(* CoDeSys 2.3.9.41 project: project_pump_station.pro *)
(* Libraries: STANDARD.LIB 4.10.05 11:14:46, IECSFC.LIB 13.4.06 15:51:28, SYSLIBTIME.LIB 26.10.21 13:46:42, SYSTASKINFO.LIB 26.10.21 13:46:42, ANALYZATION.LIB 5.10.99 09:05:06, Util.lib 18.5.10 15:14:28, SYSLIBCALLBACK.LIB 26.10.21 13:46:42 *)

(* PLC configuration (modules and I/O channels)
Fast discrete inputs [I_SIMPLE_INPUT] node 0, in %IB0 out %QB0 {ChannellName = Fast discrete inputs; Filtrationtime = 10000}
  AT %IX0.0 [BitInput] Discrete input 1 {ChannellName = Enter name}
  AT %IX0.1 [BitInput] Discrete input 2 {ChannellName = Enter name}
Discrete inputs [ID130] node 1, in %IB1 out %QB1 {ChannellName = Discrete inputs; Filtrationtime_GeneralINP = 16; PinCount = 16}
  discrete_input_first_byte AT %IB1.0 [ByteInput] discrete_input_first_byte {ChannellName = Enter name}
  discrete_input_second_byte AT %IB1.1 [ByteInput] discrete input_second_byte {ChannellName = Enter name}
Fast discrete outputs [OWEN_ID570] node 2, in %IB2 out %QB2 {ChannellName = Fast discrete outputs; SafeValueBool = FALSE; SafeValueBool = FALSE; SafeValueBool = FALSE; SafeValueBool = FALSE}
  hot_water_run_id1 AT %QX2.0 [BitOutput] Run hot water invertor drive1 {ChannellName = Enter name}
  hot_water_run_id2 AT %QX2.1 [BitOutput] Run hot water invertor drive2 {ChannellName = Enter name}
  water_supply_run_id1 AT %QX2.2 [BitOutput] Run water supply invertor drive1 {ChannellName = Enter name}
  water_supply_run_id2 AT %QX2.3 [BitOutput] Run water supply invertor drive2 {ChannellName = Enter name}
Discrete outputs [ID131] node 3, in %IB3 out %QB3 {ChannellName = Discrete outputs; SafeValueByte = 0; SafeValueByte = 0; SafeValueByteM = 0; PinCount = 24}
  AT %QB3.0 [ByteOutput] 8 discrete outputs {ChannellName = Enter name}
  AT %QB3.1 [ByteOutput] 8 discrete outputs {ChannellName = Enter name}
Special input [ID103] node 4, in %IB4 out %QB4 {ChannellName = Special input}
  AT %IX4.0 [BitInput] Special input {ChannellName = Enter name}
Special output [ID104] node 5, in %IB5 out %QB5 {ChannellName = Special output}
  AT %QX5.0 [BitOutput] Special output {ChannellName = Enter name}
ModBus (Master) [MODBUS_MASTER_ID450] node 6, in %IB6 out %QB6 {ChannellName = ModBus (Master); Visibility = No}
  AT %QD6.0 [DWordOutput] Last address {ChannellName = Enter name}
  AT %QW6.1 [WordOutput] Last error {ChannellName = Enter name}
  RS-485-1 [COM1_USART] node 0, in %IB6.0 out %QB6.0 {ChannellName = RS-485-1; CommunicationSpeed = 115200; Parity = NO PARITY CHECK; BitLength = 8 bits; StopLength = One stop bit; InterfaceType = RS485; FrameOriented = RTU; Timeout = 0; Visibility = No}
AT %QB6.1.0 [ComChannel] Command (0xff - Start) {ChannellName = Enter name}
Real input module [ID2007] node 0, in %IB6.1.0 out %QB6.1.0 {ChannellName = float input module; ModbusAddress = 4; Command_read_regs = Read holding Registers  (0x03); Visibility = No}
  input_pressure_hw AT %QD6.1.0.0 [FloatOutput] {ChannellName = Enter name}
Register input module [ID2003] node 1, in %IB6.1.1 out %QB6.1.1 {ChannellName = Register input module; ModbusAddress = 2; Command_read_regs = Read holding Registers  (0x03); Visibility = No}
  error_input_pressure_hw AT %QW6.1.1.0 [WordOutput] {ChannellName = Enter name}
Real input module [ID2007] node 2, in %IB6.1.2 out %QB6.1.2 {ChannellName = float input module; ModbusAddress = 10; Command_read_regs = Read holding Registers  (0x03); Visibility = No}
  output_pressure_hw AT %QD6.1.2.0 [FloatOutput] {ChannellName = Enter name}
Register input module [ID2003] node 3, in %IB6.1.3 out %QB6.1.3 {ChannellName = Register input module; ModbusAddress = 8; Command_read_regs = Read holding Registers  (0x03); Visibility = No}
  error_output_pressure_hw AT %QW6.1.3.0 [WordOutput] {ChannellName = Enter name}
Real input module [ID2007] node 4, in %IB6.1.4 out %QB6.1.4 {ChannellName = float input module; ModbusAddress = 16; Command_read_regs = Read holding Registers  (0x03); Visibility = No}
  input_pressure_ws AT %QD6.1.4.0 [FloatOutput] {ChannellName = Enter name}
Register input module [ID2003] node 5, in %IB6.1.5 out %QB6.1.5 {ChannellName = Register input module; ModbusAddress = 14; Command_read_regs = Read holding Registers  (0x03); Visibility = No}
  error_input_pressure_ws AT %QW6.1.5.0 [WordOutput] {ChannellName = Enter name}
Real input module [ID2007] node 6, in %IB6.1.6 out %QB6.1.6 {ChannellName = float input module; ModbusAddress = 22; Command_read_regs = Read holding Registers  (0x03); Visibility = No}
  output_pressure_ws AT %QD6.1.6.0 [FloatOutput] {ChannellName = Enter name}
Register input module [ID2003] node 7, in %IB6.1.7 out %QB6.1.7 {ChannellName = Register input module; ModbusAddress = 20; Command_read_regs = Read holding Registers  (0x03); Visibility = No}
  error_output_pressure_ws AT %QW6.1.7.0 [WordOutput] {ChannellName = Enter name}
AT %QD7.0 [DWordOutput] Last address {ChannellName = Enter name}
AT %QW7.1 [WordOutput] Last error {ChannellName = Enter name}
RS-485-1 [COM1_USART] node 0, in %IB7.0 out %QB7.0 {ChannellName = RS-485-1; CommunicationSpeed = 115200; Parity = NO PARITY CHECK; BitLength = 8 bits; StopLength = One stop bit; InterfaceType = RS485; FrameOriented = ASCII; Timeout = 0; Visibility = No}
Universal Modbus device [ID2000] node 1, in %IB7.1 out %QB7.1 {ChannellName = Universal Modbus device; ModuleIP = 10:0:0:223; ServiceTimeout = 150; TCPport = 502; NetMode = Serial; ModuleSlaveAddress = 1; RequestType = By poll time; PeriodOfService = 100; Visibility = No; RepeatCounter = 0; ByteSequence = Trace_mode}
  AT %QB7.1.0 [ComChannel] Command (0xff - Start) {ChannellName = Enter name}
output_value_hw_id1 AT %QW7.1.0.0 [WordOutput] {ChannellName = Enter name}
Register output module [ID2004] node 1, in %IB7.1.1 out %QB7.1.1 {ChannellName = Register; ModbusAddress = 0; Command_write_one_reg = Preset singl register (0x06); Visibility = No}
  output_value_hw_id2 AT %QW7.1.1.0 [WordOutput] {ChannellName = Enter name}
Register output module [ID2004] node 2, in %IB7.1.2 out %QB7.1.2 {ChannellName = Register; ModbusAddress = 0; Command_write_one_reg = Preset singl register (0x06); Visibility = No}
  output_value_ws_id1 AT %QW7.1.2.0 [WordOutput] {ChannellName = Enter name}
Register output module [ID2004] node 3, in %IB7.1.3 out %QB7.1.3 {ChannellName = Register; ModbusAddress = 0; Command_write_one_reg = Preset singl register (0x06); Visibility = No}
  output_value_ws_id2 AT %QW7.1.3.0 [WordOutput] {ChannellName = Enter name}
RS-232 [COM2_USART] node 0, in %IB8.0.0 out %QB8.0.0 {ChannellName = RS-232; CommunicationSpeed = 115200; Parity = NO PARITY CHECK; BitLength = 8 bits; StopLength = One stop bit; InterfaceType = RS232; FrameOriented = ASCII; Timeout = 0; Visibility = No}
8 bits [8Bit] node 1, in %IB8.1 out %QB8.1 {ChannellName = 8 bit}
  AT %QB8.1.0 [ByteOutput] {ChannellName = Enter name}
Float [Float] node 2, in %IB8.2 out %QB8.2 {ChannellName = float}
  hot_water_set_point_PID AT %QD8.2.0 [FloatOutput] {ChannellName = Enter name}
Float [Float] node 3, in %IB8.3 out %QB8.3 {ChannellName = float}
  water_supply_set_point_PID AT %QD8.3.0 [FloatOutput] {ChannellName = Enter name}
Float [Float] node 4, in %IB8.4 out %QB8.4 {ChannellName = float}
  P_hot_water AT %QD8.4.0 [FloatOutput] {ChannellName = Enter name}
Float [Float] node 5, in %IB8.5 out %QB8.5 {ChannellName = float}
  I_hot_water AT %QD8.5.0 [FloatOutput] {ChannellName = Enter name}
Float [Float] node 6, in %IB8.6 out %QB8.6 {ChannellName = float}
  D_hot_water AT %QD8.6.0 [FloatOutput] {ChannellName = Enter name}
Float [Float] node 7, in %IB8.7 out %QB8.7 {ChannellName = float}
  water_supply_P AT %QD8.7.0 [FloatOutput] {ChannellName = Enter name}
Float [Float] node 8, in %IB8.8 out %QB8.8 {ChannellName = float}
  water_supply_I AT %QD8.8.0 [FloatOutput] {ChannellName = Enter name}
Float [Float] node 9, in %IB8.9 out %QB8.9 {ChannellName = float}
  water_supply_D AT %QD8.9.0 [FloatOutput] {ChannellName = Enter name}
Float [Float] node 10, in %IB8.10 out %QB8.10 {ChannellName = float}
  hw_pressure_range_min AT %QD8.10.0 [FloatOutput] {ChannellName = Enter name}
Float [Float] node 11, in %IB8.11 out %QB8.11 {ChannellName = float}
  hw_pressure_range_max AT %QD8.11.0 [FloatOutput] {ChannellName = Enter name}
Float [Float] node 12, in %IB8.12 out %QB8.12 {ChannellName = float}
  water_supply_pressure_range_min AT %QD8.12.0 [FloatOutput] {ChannellName = Enter name}
Float [Float] node 13, in %IB8.13 out %QB8.13 {ChannellName = float}
  water_supply_pressure_range_max AT %QD8.13.0 [FloatOutput] {ChannellName = Enter name}
Float [Float] node 14, in %IB8.14 out %QB8.14 {ChannellName = float}
  hw_value_manual_frequency_id1 AT %QD8.14.0 [FloatOutput] {ChannellName = Enter name}
Float [Float] node 15, in %IB8.15 out %QB8.15 {ChannellName = float}
  hw_value_manual_frequency_id2 AT %QD8.15.0 [FloatOutput] {ChannellName = Enter name}
Float [Float] node 16, in %IB8.16 out %QB8.16 {ChannellName = float}
  water_supply_manual_frequency_id1 AT %QD8.16.0 [FloatOutput] {ChannellName = Enter name}
Float [Float] node 17, in %IB8.17 out %QB8.17 {ChannellName = float}
  water_supply_manual_frequency_id2 AT %QD8.17.0 [FloatOutput] {ChannellName = Enter name}
*)

(* Data type in Types data Analog_module/AnalogInputChannel *)
TYPE CAN_AnalogInputChannel :
STRUCT
	current_value: REAL;
	error_message: STRING(79);
END_STRUCT
END_TYPE

(* Data type in Types data SP310 *)
TYPE CAN_In_RS232_SP310 :
STRUCT
	pressure_input: REAL;
	pressure_output: REAL;
	status_run_invertor_drive1: BOOL;
	status_run_invertor_drive2: BOOL;
	status_alarm_invertor_drive1: BOOL;
	status_alarm_invertor_drive2: BOOL;
	PID_value: REAL;
END_STRUCT
END_TYPE

(* Data type in Types data Analog_module *)
TYPE CAN_in_RS485_Analog_module :
STRUCT

END_STRUCT
END_TYPE

(* Data type in Types data SP310 *)
TYPE CAN_Out_RS232_SP310 :
STRUCT
	auto_PID_enable: BOOL;
	cycle_enable: BOOL;
	cascade_enable: BOOL;
	set_point: REAL;
	P: REAL;
	I: REAL;
	D: REAL;
	value_manual_invertor_drive1: REAL;
	value_manual_invertor_drive2: REAL;
	pressure_range_min: REAL;
	pressure_range_max: REAL;

END_STRUCT
END_TYPE

(* Data type in ClassesProject/AnalogIModule/AnalogInputModule/AnalogInputChannel *)
TYPE classAnalogInputChannel :
STRUCT
	set_channel:classParamsValueScaling;
	value: REAL;
	error_code: WORD;
END_STRUCT
END_TYPE

(* Data type in ClassesProject/AnalogIModule/AnalogInputModule *)
TYPE classAnalogInputModule :
STRUCT
	channel1:classAnalogInputChannel;
	channel2:classAnalogInputChannel;
	channel3:classAnalogInputChannel;
	channel4:classAnalogInputChannel;
	channel5:classAnalogInputChannel;
	channel6:classAnalogInputChannel;
	channel7:classAnalogInputChannel;
	channel8:classAnalogInputChannel;
END_STRUCT
END_TYPE

(* Data type in ClassesProject/AnalogIModule/AnalogOutputModule/AnalogOutputChannel *)
TYPE classAnalogOutputChannel :
STRUCT
	register_value: WORD;
END_STRUCT
END_TYPE

(* Data type in ClassesProject/AnalogIModule/AnalogOutputModule *)
TYPE classAnalogOutputModule :
STRUCT
	channel1:classAnalogOutputChannel;
	channel2:classAnalogOutputChannel;
	channel3:classAnalogOutputChannel;
	channel4:classAnalogOutputChannel;
	channel5:classAnalogOutputChannel;
	channel6:classAnalogOutputChannel;
	channel7:classAnalogOutputChannel;
	channel8:classAnalogOutputChannel;
END_STRUCT
END_TYPE

(* Data type in ClassesProject/PLC_110_32_m2/DiscreteInputs/DiscreteInputByte *)
TYPE classDiscreteInputByte :
STRUCT
	Bit1:BOOL;
	Bit2:BOOL;
	Bit3:BOOL;
	Bit4:BOOL;
	Bit5:BOOL;
	Bit6:BOOL;
	Bit7:BOOL;
	Bit8:BOOL;
END_STRUCT
END_TYPE

(* Data type in ClassesProject/PLC_110_32_m2/DiscreteInputs *)
TYPE classDiscreteInputs :
STRUCT
	first_byte:classDiscreteInputByte;
	second_byte:classDiscreteInputByte;
END_STRUCT
END_TYPE

(* Data type in ClassesProject/PLC_110_32_m2/DiscreteOutputs/DiscreteOutputByte *)
TYPE classDiscreteOutputByte :
STRUCT
	Bit1:BOOL;
	Bit2:BOOL;
	Bit3:BOOL;
	Bit4:BOOL;
	Bit5:BOOL;
	Bit6:BOOL;
	Bit7:BOOL;
	Bit8:BOOL;
END_STRUCT
END_TYPE

(* Data type in ClassesProject/PLC_110_32_m2/DiscreteOutputs *)
TYPE classDiscreteOutputs :
STRUCT
	first_byte:classDiscreteOutputByte;
	second_byte:classDiscreteOutputByte;
END_STRUCT
END_TYPE

(* Data type in ClassesProject/PLC_110_32_m2/DiscreteInputs *)
TYPE classFastDiscreteInputs :
STRUCT
	Bit1:BOOL;
	Bit2:BOOL;
END_STRUCT
END_TYPE

(* Data type in ClassesProject/PLC_110_32_m2/DiscreteOutputs *)
TYPE classFastDiscreteOutputs :
STRUCT
	Bit1:BOOL;
	Bit2:BOOL;
	Bit3:BOOL;
	Bit4:BOOL;
END_STRUCT
END_TYPE

(* Data type in ClassesProject/InfoMessages/InfoAnalogInputModule/InfoAnalogInputChannel *)
TYPE classInfoAnalogInputChannel :
STRUCT
	current_value:REAL;
	measure:REAL;
	error_message:STRING(79);
END_STRUCT
END_TYPE

(* Data type in ClassesProject/InfoMessages/InfoAnalogInputModule *)
TYPE classInfoAnalogInputModule :
STRUCT
	channel1:classInfoAnalogInputChannel;
	channel2:classInfoAnalogInputChannel;
	channel3:classInfoAnalogInputChannel;
	channel4:classInfoAnalogInputChannel;
	channel5:classInfoAnalogInputChannel;
	channel6:classInfoAnalogInputChannel;
	channel7:classInfoAnalogInputChannel;
	channel8:classInfoAnalogInputChannel;
END_STRUCT
END_TYPE

(* Data type in ClassesProject/InfoMessages *)
TYPE classInfoCycle :
STRUCT
	run_timer: BOOL; (* статус работы таймера *)
	working_time: TIME; (*  время работы таймера *)
END_STRUCT
END_TYPE

(* Data type in ClassesProject/InfoMessages/InfoInvertorDrive *)
TYPE classInfoInvertorDrive :
STRUCT
	status_run:STRING(79);
	status_alarm:STRING(79);
	frequency:REAL;
END_STRUCT
END_TYPE

(* Data type in ClassesProject/InfoMessages *)
TYPE classInfoMessage :
STRUCT
	working_time: TIME;
	time_left: TIME;
END_STRUCT
END_TYPE

(* Data type in ClassesProject/InfoMessages/InfoPID *)
TYPE classInfoPid :
STRUCT
	out_value:REAL:=0;
	limits_active:BOOL:=FALSE;
	overflow:BOOL:=FALSE;
END_STRUCT
END_TYPE

(* Data type in ClassesProject/InvertorDrive *)
TYPE classInvertorDrive :
STRUCT
	discrete_inputs:classInvertorDriveDiscreteInputs;
	discrete_outputs:classInvertorDriveDiscreteOutputs;
	analog_input:classInvertorDriveAnalogInputs;
	analog_output:classInvertorDriveAnalogOutputs;
	set:classSetInvertorDrive;
	min_frequency:INT;
	max_frequency:INT;
	set_frequency:REAL;
	real_frequency:REAL;(* значение с аналогового выхода частотника *)
END_STRUCT
END_TYPE

(* Data type in ClassesProject/InvertorDrive *)
TYPE classInvertorDriveAnalogInputs :
STRUCT
	set_frequency:REAL;
END_STRUCT
END_TYPE

(* Data type in ClassesProject/InvertorDrive *)
TYPE classInvertorDriveAnalogOutputs :
STRUCT
	out_frequency:REAL;
END_STRUCT
END_TYPE

(* Data type in ClassesProject/InvertorDrive *)
TYPE classInvertorDriveDiscreteInputs :
STRUCT
	start:BOOL;
	reset_fault:BOOL;
END_STRUCT
END_TYPE

(* Data type in ClassesProject/InvertorDrive *)
TYPE classInvertorDriveDiscreteOutputs :
STRUCT
	status_run:BOOL;
	status_alarm:BOOL;
END_STRUCT
END_TYPE

(* Data type in ClassesProject/classesFunction *)
TYPE classParamsValueScaling :
STRUCT
	in_min: REAL:=0;
	in_max: REAL:=100;
	out_min: REAL:=0;
	out_max: REAL:=100;
END_STRUCT
END_TYPE

(* Data type in ClassesProject/PLC_110_32_m2 *)
TYPE classPLC110_32 :
STRUCT
	fast_discrete_inputs:classFastDiscreteInputs;
	discrete_inputs:classDiscreteInputs;
	special_input:classSpecialInput;
	fast_discrete_outputs:classFastDiscreteOutputs;
	discrete_output:classDiscreteOutputs;
	special_output:classSpecialOutput;
END_STRUCT
END_TYPE

(* Data type in ClassesProject/InfoMessages/PLC/110_32_m2 *)
TYPE classPLC32m2StatusInputs :
STRUCT
	fast_inputs:classFastDiscreteInputs;
	discrete_inputs:classDiscreteInputs;
	special_input:classSpecialInput;
END_STRUCT
END_TYPE

(* Data type in ClassesProject/InfoMessages/PLC/110_32_m2 *)
TYPE classPLC32m2StatusOutputs :
STRUCT
	fast_outputs:classFastDiscreteOutputs;
	discrete_outputs:classDiscreteOutputs;
	special_output:classSpecialOutput;
END_STRUCT
END_TYPE

(* Data type in ClassesProject/SP310/PumpStationSettings *)
TYPE classPumpStation :
STRUCT
	source:STRING(2);
	pump1:BOOL;
	pump2:BOOL;
	P:REAL;
	I:REAL;
	D:REAL;
	set_point:REAL;
	cycle_enable:BOOL;
	cascade_enable:BOOL;
	seconds_cycle: TIME;
	minutes_cycle: TIME;
	hours_cycle: TIME;
END_STRUCT
END_TYPE

(* Data type in ClassesProject/AnalogIModule/AnalogInputModule/SetAnalogInputsModule/SetAnalogInputChannel *)
TYPE classSetAnalogInputChannel :
STRUCT
	(* Конфигурационные параметры канала модуля. см. инструкцию прибора: приложение. таблица В.2 *)
	(* Границы АЦП и значения по умолчанию: для датчика 4-20mA  *)
	ain_l: REAL := 0;  (* Параметр Ain.L *)
	ain_h: REAL := 1000;  (* Параметр Ain.H *)
	analog_min_value: REAL := 4;  (* Диапазон нижней границы датчика давления *)
	analog_max_value: REAL := 20;  (* Диапазон верхней границы датчика давления *)
END_STRUCT
END_TYPE

(* Data type in ClassesProject/AnalogIModule/AnalogInputModule/SetAnalogInputsModule *)
TYPE classSetAnalogInputsModule :
STRUCT
	ch1_set:classSetAnalogInputChannel;
	ch2_set:classSetAnalogInputChannel;
	ch3_set:classSetAnalogInputChannel;
	ch4_set:classSetAnalogInputChannel;
	ch5_set:classSetAnalogInputChannel;
	ch6_set:classSetAnalogInputChannel;
	ch7_set:classSetAnalogInputChannel;
	ch8_set:classSetAnalogInputChannel;
END_STRUCT
END_TYPE

(* Data type in ClassesProject/InvertorDrive/SetInvertorDrive/SetAutoInvertorDrive *)
TYPE classSetAutoInvertorDrive :
STRUCT
	auto:BOOL:=FALSE;
	direct_logic:BOOL:=TRUE;  (* флаг прямого/обратного управления; при обратном управлении если значение контролируемой величины ниже уставки, выходная частота уменьшается, и наоборот*)
	set_point:REAL:=0;  (* уставка, задается в единицах измерения контролируемой величины *)
	value:REAL:=0;  (* текущее значение контролируемой величины, получаемое с датчика *)
	P:REAL:=2;  (* Пропорциональный коэффициент регулятора, при увеличении выход регулятора изменяется быстрее*)
	I:INT:=10;  (* Интегральный коэффичиент регулятора, время в секундах *)
	D:INT:=0;  (* Дифференциальный коэффичиент регулятора, время в секундах *)
END_STRUCT
END_TYPE

(* Data type in ClassesProject/InvertorDrive/SetInvertorDrive *)
TYPE classSetInvertorDrive :
STRUCT
	set_auto:classSetAutoInvertorDrive;
	set_frequency:classSetLimitFrequency;
END_STRUCT
END_TYPE

(* Data type in ClassesProject/Sensors/Kpi *)
TYPE classSetKpi :
STRUCT
	range:REAL;
	diff:REAL:=0.2;
END_STRUCT
END_TYPE

(* Data type in ClassesProject/InvertorDrive/SetInvertorDrive/SetLimitFrequency *)
TYPE classSetLimitFrequency :
STRUCT
	manual:REAL;  (* Hz *)
	min_range:REAL;  (* Hz *)
	max_range:REAL;  (* Hz *)
END_STRUCT
END_TYPE

(* Data type in ClassesProject/PID *)
TYPE classSetPid :
STRUCT
	actual:REAL;
	set_point:REAL;
	P:REAL;  (* Пропорциональный коэффициент регулятора, при увеличении выход регулятора изменяется быстрее*)
	I:INT;  (* Интегральный коэффичиент регулятора, время в секундах *)
	D:INT;  (* Дифференциальный коэффичиент регулятора, время в секундах *)
	Y_manual:REAL:=0;
	Y_offset:REAL;
	Y_min:REAL;
	Y_max:REAL;
	manual:BOOL;
	reset:BOOL;
END_STRUCT
END_TYPE

(* Data type in ClassesProject/Sensors/PressureSensors/CurrentPressures/4-20mA *)
TYPE classSetPressureSensor4_20 :
STRUCT
	min_measure_range:REAL;
	max_measure_range:REAL;
	min_current_range:REAL:=4;
	max_current_range:REAL:=20;
END_STRUCT
END_TYPE

(* Data type in ClassesProject/SP310 *)
TYPE classSP310 :
STRUCT
	hot_water:classPumpStation;
	water_supply:classPumpStation;
END_STRUCT
END_TYPE

(* Data type in ClassesProject/PLC_110_32_m2/DiscreteInputs *)
TYPE classSpecialInput :
STRUCT
	Bit1:BOOL;
END_STRUCT
END_TYPE

(* Data type in ClassesProject/PLC_110_32_m2/DiscreteOutputs *)
TYPE classSpecialOutput :
STRUCT
	Bit1:BOOL;
END_STRUCT
END_TYPE

(* Data type in Types data InvertorDrive *)
TYPE InvertorStatusData :
STRUCT
	status_alarm: BOOL;
	status_run: BOOL;
END_STRUCT
END_TYPE

(* POU PLC_PRG, CFC *)
PROGRAM PLC_PRG
VAR
	info_channel:classInfoAnalogInputChannel;

	info2: classInfoAnalogInputChannel;
	channel1: AnalogInputChannel;
	sensor1: SetCurrentSensorPressure_4_20;
	Settings1: ParamsAnalogInputChannel;
	PLC: PLC110_32m2;
	PLCstatus_intputs:classPLC32m2StatusInputs;
	Kpi35_HW: Kpi;
	Kpi36_HW: Kpi;


	HW_discrete_inputs_id1: InvertorDriveInputs;
	HW_discrete_outputs_id1: InvertorDriveOutputs;
	HW_id1: InvertorDrive;
	AinModuleSettings: SetChannelsAnalogInputsModule;
	AnalogInputsModule: MB110_8a;
	Ain_info: BOOL;
END_VAR
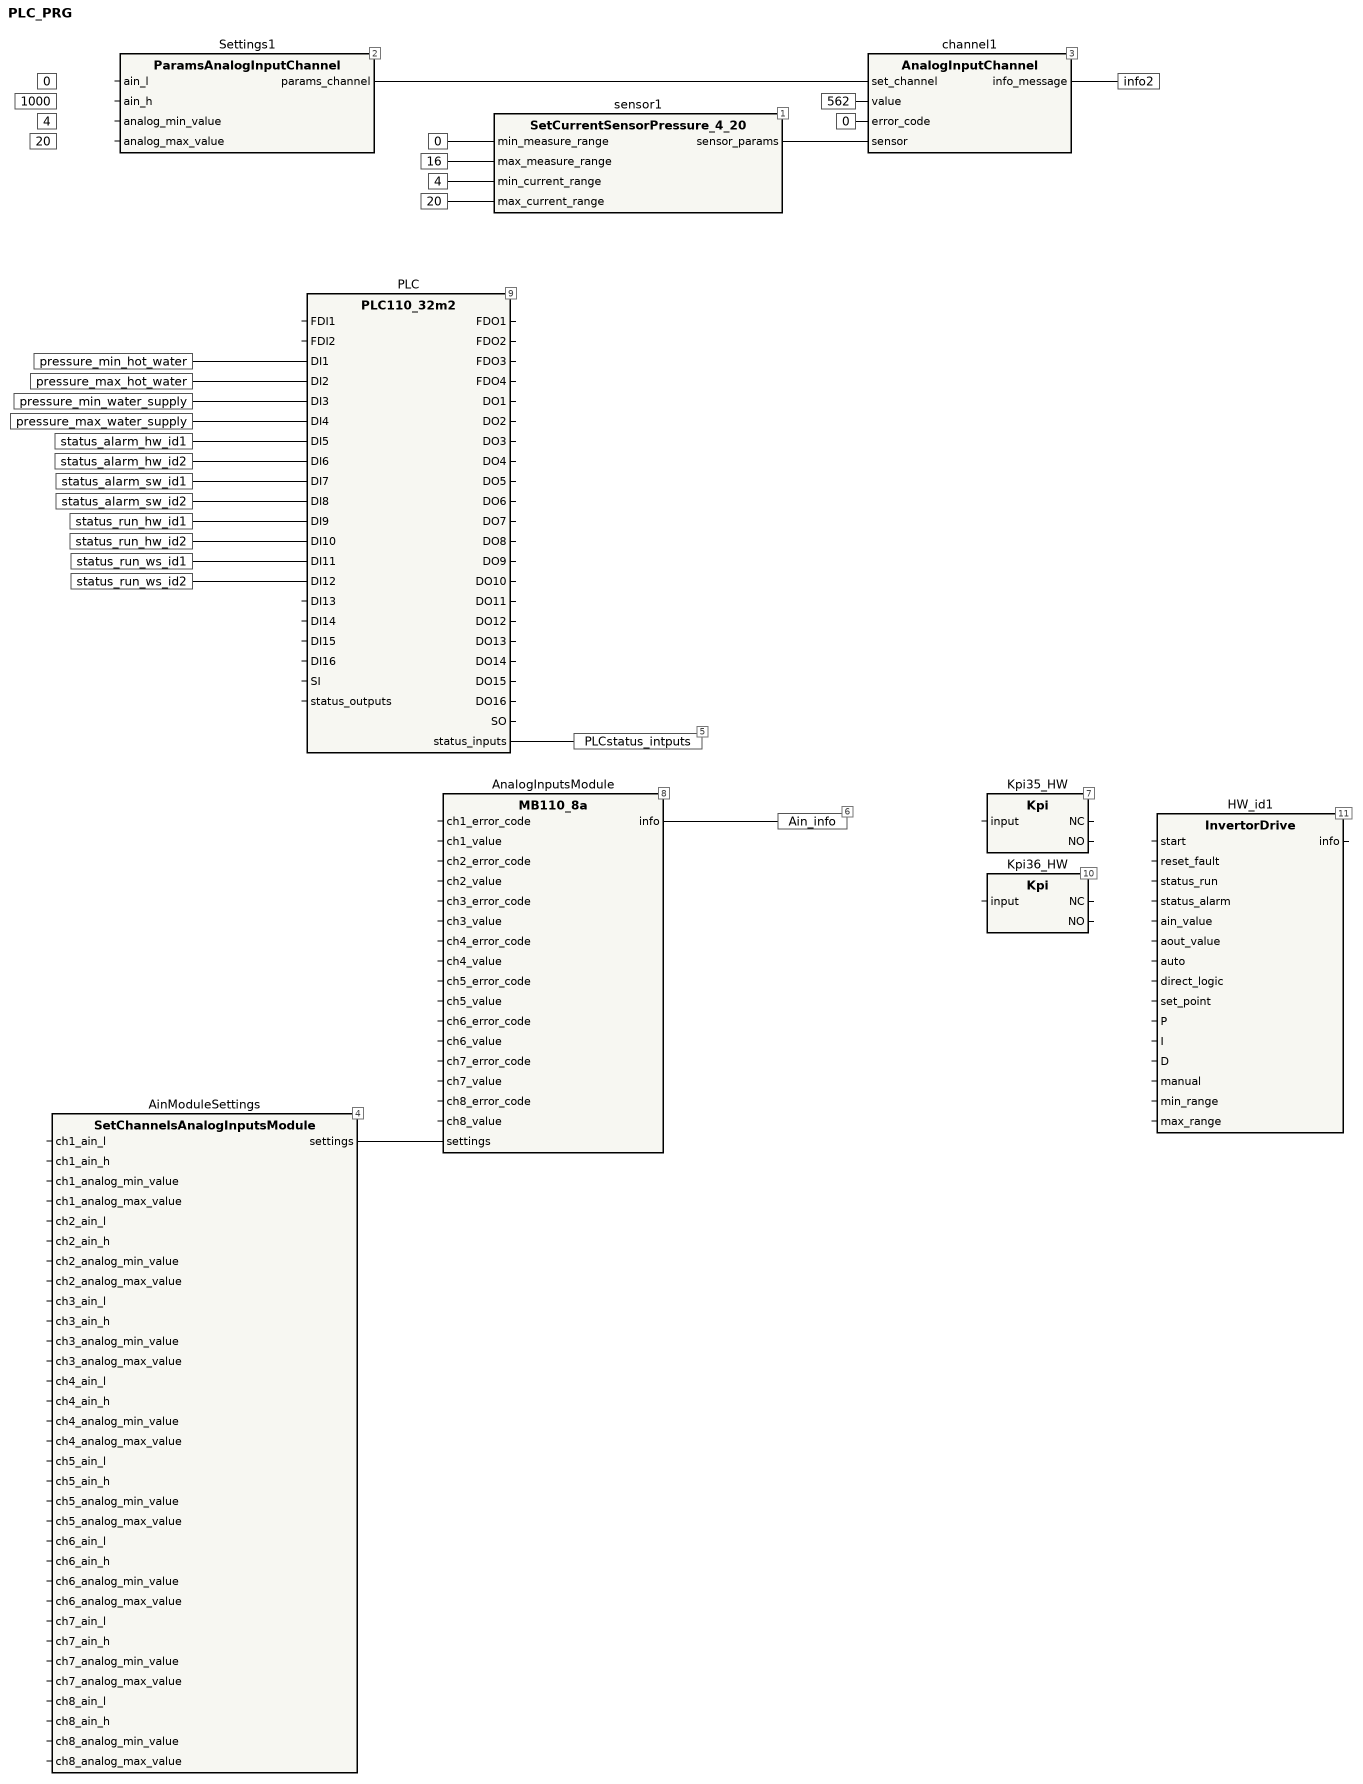
_CFC_ (* Continuous Function Chart, elements in execution order *)
unconnected input 0
unconnected input 1000
unconnected input 4
unconnected input 20
#0 info2 <= #3.info_message
#1 sensor1:SetCurrentSensorPressure_4_20(min_measure_range: 0, max_measure_range: 16, min_current_range: 4, max_current_range: 20)
#2 Settings1:ParamsAnalogInputChannel(ain_l: -, ain_h: -, analog_min_value: -, analog_max_value: -)
#3 channel1:AnalogInputChannel(set_channel: #2.params_channel, value: 562, error_code: 0, sensor: #1.sensor_params)
#4 AinModuleSettings:SetChannelsAnalogInputsModule(ch1_ain_l: -, ch1_ain_h: -, ch1_analog_min_value: -, ch1_analog_max_value: -, ch2_ain_l: -, ch2_ain_h: -, ch2_analog_min_value: -, ch2_analog_max_value: -, ch3_ain_l: -, ch3_ain_h: -, ch3_analog_min_value: -, ch3_analog_max_value: -, ch4_ain_l: -, ch4_ain_h: -, ch4_analog_min_value: -, ch4_analog_max_value: -, ch5_ain_l: -, ch5_ain_h: -, ch5_analog_min_value: -, ch5_analog_max_value: -, ch6_ain_l: -, ch6_ain_h: -, ch6_analog_min_value: -, ch6_analog_max_value: -, ch7_ain_l: -, ch7_ain_h: -, ch7_analog_min_value: -, ch7_analog_max_value: -, ch8_ain_l: -, ch8_ain_h: -, ch8_analog_min_value: -, ch8_analog_max_value: -)
#5 PLCstatus_intputs <= #9.status_inputs
#6 Ain_info <= #8.info
#7 Kpi35_HW:Kpi(input: -)
#8 AnalogInputsModule:MB110_8a(ch1_error_code: -, ch1_value: -, ch2_error_code: -, ch2_value: -, ch3_error_code: -, ch3_value: -, ch4_error_code: -, ch4_value: -, ch5_error_code: -, ch5_value: -, ch6_error_code: -, ch6_value: -, ch7_error_code: -, ch7_value: -, ch8_error_code: -, ch8_value: -, settings: #4.settings)
#9 PLC:PLC110_32m2(FDI1: -, FDI2: -, DI1: pressure_min_hot_water, DI2: pressure_max_hot_water, DI3: pressure_min_water_supply, DI4: pressure_max_water_supply, DI5: status_alarm_hw_id1, DI6: status_alarm_hw_id2, DI7: status_alarm_sw_id1, DI8: status_alarm_sw_id2, DI9: status_run_hw_id1, DI10: status_run_hw_id2, DI11: status_run_ws_id1, DI12: status_run_ws_id2, DI13: -, DI14: -, DI15: -, DI16: -, SI: -, status_outputs: -)
#10 Kpi36_HW:Kpi(input: -)
#11 HW_id1:InvertorDrive(start: -, reset_fault: -, status_run: -, status_alarm: -, ain_value: -, aout_value: -, auto: -, direct_logic: -, set_point: -, P: -, I: -, D: -, manual: -, min_range: -, max_range: -)
_END_CFC_
(* the same logic as Structured Text *)
info2 := channel1.info_message;
sensor1(min_measure_range := 0, max_measure_range := 16, min_current_range := 4, max_current_range := 20);
Settings1();
channel1(set_channel := Settings1.params_channel, value := 562, error_code := 0, sensor := sensor1.sensor_params);
AinModuleSettings();
PLCstatus_intputs := PLC.status_inputs;
Ain_info := AnalogInputsModule.info;
Kpi35_HW();
AnalogInputsModule(settings := AinModuleSettings.settings);
PLC(DI1 := pressure_min_hot_water, DI2 := pressure_max_hot_water, DI3 := pressure_min_water_supply, DI4 := pressure_max_water_supply, DI5 := status_alarm_hw_id1, DI6 := status_alarm_hw_id2, DI7 := status_alarm_sw_id1, DI8 := status_alarm_sw_id2, DI9 := status_run_hw_id1, DI10 := status_run_hw_id2, DI11 := status_run_ws_id1, DI12 := status_run_ws_id2);
Kpi36_HW();
HW_id1();
END_PROGRAM

(* POU ObjectsProject/AnalogInputsModule/AnalogInputChannel/AnalogInputChannel, ST *)
FUNCTION_BLOCK AnalogInputChannel
VAR_INPUT
	set_channel:classSetAnalogInputChannel;
	value:REAL;
	error_code:WORD;
	sensor:classSetPressureSensor4_20;
END_VAR
VAR_OUTPUT
	info_message:classInfoAnalogInputChannel;
END_VAR
VAR
	channel:classAnalogInputChannel;
END_VAR
channel.set_channel:=get_params_value_scaling(set_channel.ain_l, set_channel.ain_h, set_channel.analog_min_value, set_channel.analog_max_value);
channel.value:=value;
channel.error_code:=error_code;

info_message:=get_infos_analog_input_channel(sensor, channel);
END_FUNCTION_BLOCK

(* POU FunctionCannel/ValueScaling/get_params_value_scaling, ST *)
FUNCTION get_params_value_scaling : classParamsValueScaling
VAR_INPUT
	in_min: REAL;
	in_max: REAL;
	out_min: REAL;
	out_max: REAL;
END_VAR
VAR
END_VAR
get_params_value_scaling.in_min:=in_min;
get_params_value_scaling.in_max:=in_max;
get_params_value_scaling.out_min:=out_min;
get_params_value_scaling.out_max:=out_max;
END_FUNCTION

(* POU ClassesProject/AnalogInputsModule/AnalogInputChannel/get_infos_analog_input_channel, ST *)
FUNCTION get_infos_analog_input_channel : classInfoAnalogInputChannel
VAR_INPUT
	sensor:classSetPressureSensor4_20;
	channel:classAnalogInputChannel;
END_VAR
VAR

END_VAR
get_infos_analog_input_channel.error_message := get_error_code(channel.error_code);
IF channel.error_code = 0 THEN

	get_infos_analog_input_channel.current_value := value_scaling(channel.value, channel.set_channel);
	get_infos_analog_input_channel.measure := value_scaling(get_infos_analog_input_channel.current_value, get_params_value_scaling(sensor.min_current_range, sensor.max_current_range, sensor.min_measure_range, sensor.max_measure_range));
ELSE
	(* если модуль вернул ошибку покажем писюны *)
	get_infos_analog_input_channel.current_value := -8;
	get_infos_analog_input_channel.measure := -8;
END_IF
END_FUNCTION

(* POU ClassesProject/AnalogInputsModule/AnalogInputChannel/get_error_code, ST *)
FUNCTION get_error_code: STRING(79)
(* Функция преобразования кода ошибки регистра аналогового модуля входов *)
VAR_INPUT
	code_error: WORD;
END_VAR
VAR
	error_message: STRING(79);
END_VAR
IF code_error = 0
	THEN error_message := 'Измерение успешно';
ELSIF code_error = 61440
	THEN error_message := 'Значение заведомо неверно';
ELSIF code_error = 61446
	THEN error_message := 'Данные не готовы. Ждите результатов первого измерения.';
ELSIF code_error = 61447
	THEN error_message := 'Датчик отключен.';
ELSIF code_error = 61448
	THEN error_message := 'Велика температура свободныз концов ТП.';
ELSIF code_error = 61449
	THEN error_message := 'Мала температура свободных концов ТП.';
ELSIF code_error = 61450
	THEN error_message := 'Измеренное значение слишком велико.';
ELSIF code_error = 61451
	THEN error_message := 'Измеренное значение слишком мало.';
ELSIF code_error = 61452
	THEN error_message := 'Короткое замыкание датчика.';
ELSIF code_error = 61453
	THEN error_message := 'Обрыв датчика.';
ELSIF code_error = 61454
	THEN error_message := 'Отсутствие связи с АЦП.';
ELSIF code_error = 61455
	THEN error_message := 'Некорректный калибровочный коэффициент.';
ELSE
	error_message := 'Error not Found';
END_IF

get_error_code := error_message;
END_FUNCTION

(* POU FunctionCannel/ValueScaling/value_scaling, ST *)
FUNCTION value_scaling : REAL
(* Функция масштабирования шкалы *)
VAR_INPUT
	input_value: REAL;
	params_scales:classParamsValueScaling;
END_VAR
VAR
	A: REAL;
	B: REAL;
END_VAR
A := (params_scales.out_max - params_scales.out_min) / (params_scales.in_max - params_scales.in_min);
B := ((params_scales.out_min * params_scales.in_max) - (params_scales.out_max * params_scales.in_min)) / (params_scales.in_max - params_scales.in_min);

value_scaling := A * input_value + B;
END_FUNCTION

(* POU ObjectsProject/PressureSensors/CurrentSensors/Current_4_20/SetCurrentSensorPressure_4_20, ST *)
FUNCTION_BLOCK SetCurrentSensorPressure_4_20
VAR_INPUT
	min_measure_range:REAL;
	max_measure_range:REAL;
	min_current_range:REAL:=4;
	max_current_range:REAL:=20;
END_VAR
VAR_OUTPUT
	sensor_params:classSetPressureSensor4_20;
END_VAR
VAR
END_VAR
sensor_params.min_measure_range:=min_measure_range;
sensor_params.max_measure_range:=max_measure_range;
sensor_params.min_current_range:=min_current_range;
sensor_params.max_current_range:=max_current_range;
END_FUNCTION_BLOCK

(* POU ObjectsProject/AnalogInputsModule/AnalogInputChannel/ParamsAnalogInputChannel, ST *)
FUNCTION_BLOCK ParamsAnalogInputChannel
VAR_INPUT
	(* Конфигурационные параметры канала модуля. см. инструкцию прибора: приложение. таблица В.2 *)
	(* Границы АЦП и значения по умолчанию: для датчика 4-20mA  *)
	ain_l: REAL := 0;  (* Параметр Ain.L *)
	ain_h: REAL := 1000;  (* Параметр Ain.H *)
	analog_min_value: REAL := 4;  (* Диапазон нижней границы датчика давления *)
	analog_max_value: REAL := 20;  (* Диапазон верхней границы датчика давления *)

END_VAR
VAR_OUTPUT
	params_channel:classSetAnalogInputChannel;
END_VAR
VAR
END_VAR
params_channel.ain_l:=ain_l;
params_channel.ain_h:=ain_h;
params_channel.analog_min_value:=analog_min_value;
params_channel.analog_max_value:=analog_max_value;
END_FUNCTION_BLOCK

(* POU ObjectsProject/PLC110/32m2/PLC110_32m2, ST *)
FUNCTION_BLOCK PLC110_32m2
VAR_INPUT
	FDI1:BOOL;
	FDI2:BOOL;
	DI1:BOOL;
	DI2:BOOL;
	DI3:BOOL;
	DI4:BOOL;
	DI5:BOOL;
	DI6:BOOL;
	DI7:BOOL;
	DI8:BOOL;
	DI9:BOOL;
	DI10:BOOL;
	DI11:BOOL;
	DI12:BOOL;
	DI13:BOOL;
	DI14:BOOL;
	DI15:BOOL;
	DI16:BOOL;
	SI:BOOL;
	status_outputs:classPLC32m2StatusOutputs;
END_VAR
VAR_OUTPUT
	FDO1:BOOL;
	FDO2:BOOL;
	FDO3:BOOL;
	FDO4:BOOL;
	DO1:BOOL;
	DO2:BOOL;
	DO3:BOOL;
	DO4:BOOL;
	DO5:BOOL;
	DO6:BOOL;
	DO7:BOOL;
	DO8:BOOL;
	DO9:BOOL;
	DO10:BOOL;
	DO11:BOOL;
	DO12:BOOL;
	DO13:BOOL;
	DO14:BOOL;
	DO15:BOOL;
	DO16:BOOL;
	SO:BOOL;
	status_inputs:classPLC32m2StatusInputs;
END_VAR
VAR
	fast_inputs:classFastDiscreteInputs;
	discrete_inputs:classDiscreteInputs;
	special_input:classSpecialInput;
	fast_outputs:classFastDiscreteOutputs;
	discrete_outputs:classDiscreteOutputs;
	special_output:classSpecialOutput;
END_VAR
init;

get_status_inputs;
END_FUNCTION_BLOCK
ACTION get_status_inputs:
status_inputs.fast_inputs:=fast_inputs;
status_inputs.discrete_inputs:=discrete_inputs;
status_inputs.special_input:=special_input;
END_ACTION
ACTION init:
fast_inputs.Bit1:=FDI1;
fast_inputs.Bit2:=FDI2;

discrete_inputs.first_byte.Bit1:=DI1;
discrete_inputs.first_byte.Bit2:=DI2;
discrete_inputs.first_byte.Bit3:=DI3;
discrete_inputs.first_byte.Bit4:=DI4;
discrete_inputs.first_byte.Bit5:=DI5;
discrete_inputs.first_byte.Bit6:=DI6;
discrete_inputs.first_byte.Bit7:=DI7;
discrete_inputs.first_byte.Bit8:=DI8;
discrete_inputs.second_byte.Bit1:=DI9;
discrete_inputs.second_byte.Bit2:=DI10;
discrete_inputs.second_byte.Bit3:=DI11;
discrete_inputs.second_byte.Bit4:=DI12;
discrete_inputs.second_byte.Bit5:=DI13;
discrete_inputs.second_byte.Bit6:=DI14;
discrete_inputs.second_byte.Bit7:=DI15;
discrete_inputs.second_byte.Bit8:=DI16;

special_input.Bit1:=SI;

fast_outputs.Bit1:=FDO1;
fast_outputs.Bit2:=FDO2;
fast_outputs.Bit3:=FDO3;
fast_outputs.Bit4:=FDO4;

discrete_outputs.first_byte.Bit1:=DO1;
discrete_outputs.first_byte.Bit2:=DO2;
discrete_outputs.first_byte.Bit3:=DO3;
discrete_outputs.first_byte.Bit4:=DO4;
discrete_outputs.first_byte.Bit5:=DO5;
discrete_outputs.first_byte.Bit6:=DO6;
discrete_outputs.first_byte.Bit7:=DO7;
discrete_outputs.first_byte.Bit8:=DO8;

discrete_outputs.second_byte.Bit1:=DO9;
discrete_outputs.second_byte.Bit2:=DO10;
discrete_outputs.second_byte.Bit3:=DO11;
discrete_outputs.second_byte.Bit4:=DO12;
discrete_outputs.second_byte.Bit5:=DO13;
discrete_outputs.second_byte.Bit6:=DO14;
discrete_outputs.second_byte.Bit7:=DO15;
discrete_outputs.second_byte.Bit8:=DO16;

special_output.Bit1:=SO;
END_ACTION

(* POU ObjectsProject/PressureSensors/Kpi/Kpi, ST *)
FUNCTION_BLOCK Kpi
VAR_INPUT
	input:BOOL;  (* давление на входе *)
	(* model:INT;
	on:BOOL; *)
END_VAR
VAR_OUTPUT
	NC:BOOL; (* normal close №2 *)
	NO:BOOL; (* normal open №4 *)
END_VAR
VAR
	set:classSetKpi;
END_VAR
(* IF model = 35 THEN
	set.range:=2;
	set.diff:=0.4;
ELSIF model = 36 THEN
	set.range:= 8;
	set.diff:=0.5;
END_IF; *)

NC:=NOT input;
NO:=input;
END_FUNCTION_BLOCK

(* POU ObjectsProject/InvertorDrive/InvertorDriveInputs, ST *)
FUNCTION_BLOCK InvertorDriveInputs
VAR_INPUT
	start:BOOL;
	reset_fault:BOOL;
END_VAR
VAR_OUTPUT
	inputs:classInvertorDriveDiscreteInputs;
END_VAR
VAR
END_VAR
inputs.start:=start;
inputs.reset_fault:=reset_fault;
END_FUNCTION_BLOCK

(* POU ObjectsProject/InvertorDrive/InvertorDriveOutputs, ST *)
FUNCTION_BLOCK InvertorDriveOutputs
VAR_INPUT
	status_run:BOOL;
	status_alarm:BOOL;
END_VAR
VAR_OUTPUT
	outputs:classInvertorDriveDiscreteOutputs;
END_VAR
VAR
END_VAR
outputs.status_run:=status_run;
outputs.status_alarm:=status_alarm;
END_FUNCTION_BLOCK

(* POU ObjectsProject/InvertorDrive/InvertorDrive, ST *)
FUNCTION_BLOCK InvertorDrive
VAR_INPUT
(* discrete inputs *)
	start:BOOL:=FALSE;
	reset_fault:BOOL:=FALSE;
(* discrete outputs *)
	status_run:BOOL;
	status_alarm:BOOL;
(* analog inputs *)
	ain_value:REAL:=0;  (* mA or V *)
(* analog outputs *)
	aout_value:REAL:=0;
(* PID settings *)
	auto:BOOL;
	direct_logic:BOOL:=TRUE;  (* флаг прямого/обратного управления; при обратном управлении если значение контролируемой величины ниже уставки, выходная частота уменьшается, и наоборот*)
	set_point:REAL:=0;  (* уставка, задается в единицах измерения контролируемой величины *)
	(* value:REAL;  текущее значение контролируемой величины, получаемое с датчика *)
	P:REAL:=2;  (* Пропорциональный коэффициент регулятора, при увеличении выход регулятора изменяется быстрее*)
	I:INT:=10;  (* Интегральный коэффичиент регулятора, время в секундах *)
	D:INT:=0;  (* Дифференциальный коэффичиент регулятора, время в секундах *)

(* limit work frequency *)
	manual:REAL:=0;(*Hz*)
	min_range:REAL:=15;  (*Hz*)
	max_range:REAL:=50;  (*Hz*)
END_VAR
VAR_OUTPUT
	info:classInfoInvertorDrive;
END_VAR
VAR
	invertor_drive:classInvertorDrive;
       set_auto:classSetAutoInvertorDrive;
	set_frequency: classSetLimitFrequency;
	set_pid:classSetPid;
	regulator_pid:PID;
	overflow:BOOL;

	results_pid: classInfoPid;
	no_owerflow: TON;

	discrete_inputs: classInvertorDriveDiscreteInputs;
	discrete_outputs: classInvertorDriveDiscreteOutputs;
	None_pid: classInfoPid;
	analog_inputs: classInvertorDriveAnalogInputs;
END_VAR
init;

get_value_out_frequency;

get_infomessage;
END_FUNCTION_BLOCK
ACTION get_infoMessage:
info.frequency:=results_pid.out_value;  (* Hz *)

IF discrete_outputs.status_alarm THEN
	info.status_alarm:='Авария частотного преобразователя!';
ELSE
	info.status_alarm:='Аварий нет';
END_IF;

IF discrete_outputs.status_run THEN
	info.status_run:='Запущен';
ELSE
	info.status_run:='Остановлен';
END_IF;
END_ACTION
ACTION get_value_out_frequency:
IF discrete_inputs.start THEN
	analog_inputs:=invertor_drive.analog_input;
	set_auto:=invertor_drive.set.set_auto;
	set_frequency:=invertor_drive.set.set_frequency;

	overflow:=FALSE; (* сюда прикрутить таймер цикла *)

	set_pid:=get_set_pid(set_auto.direct_logic,	set_auto.value, set_auto.set_point, set_auto.P, set_auto.I, set_auto.D, set_frequency.manual, 0, set_frequency.min_range, set_frequency.max_range, NOT set_auto.auto, overflow);
	results_pid:=get_PID(set_pid);
ELSE
(* если выключено возвращаем нули *)
	results_pid:=None_pid;
END_IF;
END_ACTION
ACTION init:
invertor_drive.analog_input.set_frequency:=ain_value;
invertor_drive.analog_output.out_frequency:=aout_value;

invertor_drive.discrete_inputs.start:=start;
invertor_drive.discrete_inputs.reset_fault:=reset_fault;

invertor_drive.discrete_outputs.status_run:=status_run;
invertor_drive.discrete_outputs.status_alarm:=status_alarm;

invertor_drive.set.set_frequency.min_range:=min_range;
invertor_drive.set.set_frequency.max_range:=max_range;

invertor_drive.set.set_auto.auto:=auto;
invertor_drive.set.set_auto.direct_logic:=direct_logic;
invertor_drive.set.set_auto.set_point:=set_point;
invertor_drive.set.set_auto.value:=ain_value;
invertor_drive.set.set_auto.P:=P;
invertor_drive.set.set_auto.I:=I;
invertor_drive.set.set_auto.D:=D;

invertor_drive.set.set_frequency.manual:=manual;
invertor_drive.set.set_frequency.min_range:=min_range;
invertor_drive.set.set_frequency.max_range:=max_range;

discrete_inputs:=invertor_drive.discrete_inputs;
discrete_outputs:=invertor_drive.discrete_outputs;
END_ACTION

(* POU ObjectsProject/PID_regulator/get_set_pid, ST *)
FUNCTION get_set_pid : classSetPid
VAR_INPUT
	direct_logic:BOOL;
	actual:REAL;
	set_point:REAL;
	P:REAL;  (* Пропорциональный коэффициент регулятора, при увеличении выход регулятора изменяется быстрее*)
	I:INT;  (* Интегральный коэффичиент регулятора, время в секундах *)
	D:INT;  (* Дифференциальный коэффичиент регулятора, время в секундах *)
	Y_manual:REAL:=0;
	Y_offset:REAL:=0;
	Y_min:REAL;
	Y_max:REAL;
	manual:BOOL:=TRUE;
	reset:BOOL:=FALSE;
END_VAR
VAR
END_VAR
IF direct_logic = TRUE THEN
	get_set_pid.actual:=actual;
	get_set_pid.set_point:=set_point;
ELSE
	get_set_pid.actual:=set_point;
	get_set_pid.set_point:=actual;
END_IF;

get_set_pid.P:=P;
get_set_pid.I:=I;
get_set_pid.D:=D;
get_set_pid.Y_manual:=Y_manual;
get_set_pid.Y_offset:=Y_offset;
get_set_pid.Y_min:=Y_min;
get_set_pid.Y_max:=Y_max;
get_set_pid.manual:=manual;
get_set_pid.reset:=reset;
END_FUNCTION

(* POU ObjectsProject/PID_regulator/get_PID, ST *)
FUNCTION get_PID : classInfoPid
VAR_INPUT
	set:classSetPid;
END_VAR
VAR
	regulator:PID;
END_VAR
regulator.ACTUAL:=set.actual;
regulator.SET_POINT:=set.set_point;
regulator.KP:=set.P;
regulator.TN:=set.I;
regulator.TV:=set.D;
regulator.Y_MANUAL:=set.Y_manual;
regulator.Y_OFFSET:=set.Y_offset;
regulator.Y_MIN:=set.Y_min;
regulator.Y_MAX:=set.Y_max;
regulator.MANUAL:=set.manual;
regulator.RESET:=set.reset;

get_PID.out_value:=regulator.Y;
get_PID.limits_active:=regulator.LIMITS_ACTIVE;
get_PID.overflow:=regulator.OVERFLOW;
END_FUNCTION

(* POU ObjectsProject/AnalogInputsModule/MB110_8a/SetChannelsAnalogInputsModule, ST *)
FUNCTION_BLOCK SetChannelsAnalogInputsModule
VAR_INPUT
	(* Конфигурационные параметры канала модуля. см. инструкцию прибора: приложение. таблица В.2 *)
	(* Границы АЦП и значения по умолчанию: для датчика 4-20mA  *)

	ch1_ain_l: REAL := 0;  (* Параметр Ain.L *)
	ch1_ain_h: REAL := 100;  (* Параметр Ain.H *)
	ch1_analog_min_value: REAL := 4;  (* Диапазон нижней границы датчика *)
	ch1_analog_max_value: REAL := 20;  (* Диапазон верхней границы датчика *)

	ch2_ain_l: REAL := 0;  (* Параметр Ain.L *)
	ch2_ain_h: REAL := 100;  (* Параметр Ain.H *)
	ch2_analog_min_value: REAL := 4;  (* Диапазон нижней границы датчика *)
	ch2_analog_max_value: REAL := 20;  (* Диапазон верхней границы датчика *)

	ch3_ain_l: REAL := 0;  (* Параметр Ain.L *)
	ch3_ain_h: REAL := 100;  (* Параметр Ain.H *)
	ch3_analog_min_value: REAL := 4;  (* Диапазон нижней границы датчика *)
	ch3_analog_max_value: REAL := 20;  (* Диапазон верхней границы датчика *)

	ch4_ain_l: REAL := 0;  (* Параметр Ain.L *)
	ch4_ain_h: REAL := 100;  (* Параметр Ain.H *)
	ch4_analog_min_value: REAL := 4;  (* Диапазон нижней границы датчика *)
	ch4_analog_max_value: REAL := 20;  (* Диапазон верхней границы датчика *)

	ch5_ain_l: REAL := 0;  (* Параметр Ain.L *)
	ch5_ain_h: REAL := 100;  (* Параметр Ain.H *)
	ch5_analog_min_value: REAL := 4;  (* Диапазон нижней границы датчика *)
	ch5_analog_max_value: REAL := 20;  (* Диапазон верхней границы датчика *)

	ch6_ain_l: REAL := 0;  (* Параметр Ain.L *)
	ch6_ain_h: REAL := 100;  (* Параметр Ain.H *)
	ch6_analog_min_value: REAL := 4;  (* Диапазон нижней границы датчика *)
	ch6_analog_max_value: REAL := 20;  (* Диапазон верхней границы датчика *)

	ch7_ain_l: REAL := 0;  (* Параметр Ain.L *)
	ch7_ain_h: REAL := 100;  (* Параметр Ain.H *)
	ch7_analog_min_value: REAL := 4;  (* Диапазон нижней границы датчика *)
	ch7_analog_max_value: REAL := 20;  (* Диапазон верхней границы датчика *)

	ch8_ain_l: REAL := 0;  (* Параметр Ain.L *)
	ch8_ain_h: REAL := 100;  (* Параметр Ain.H *)
	ch8_analog_min_value: REAL := 4;  (* Диапазон нижней границы датчика *)
	ch8_analog_max_value: REAL := 20;  (* Диапазон верхней границы датчика *)
END_VAR
VAR_OUTPUT
	settings:classSetAnalogInputsModule;
END_VAR
VAR

END_VAR
settings.ch1_set.ain_l:=ch1_ain_l;
settings.ch1_set.ain_h:=ch1_ain_h;
settings.ch1_set.analog_min_value:=ch1_analog_min_value;
settings.ch1_set.analog_max_value:=ch1_analog_max_value;
get_settings;
END_FUNCTION_BLOCK
ACTION get_settings:
settings.ch1_set.ain_l:=ch1_ain_l;
settings.ch1_set.ain_h:=ch1_ain_h;
settings.ch1_set.analog_min_value:=ch1_analog_min_value;
settings.ch1_set.analog_max_value:=ch1_analog_max_value;

settings.ch2_set.ain_l:=ch2_ain_l;
settings.ch2_set.ain_h:=ch2_ain_h;
settings.ch2_set.analog_min_value:=ch2_analog_min_value;
settings.ch2_set.analog_max_value:=ch2_analog_max_value;

settings.ch3_set.ain_l:=ch3_ain_l;
settings.ch3_set.ain_h:=ch3_ain_h;
settings.ch3_set.analog_min_value:=ch3_analog_min_value;
settings.ch3_set.analog_max_value:=ch3_analog_max_value;

settings.ch4_set.ain_l:=ch4_ain_l;
settings.ch4_set.ain_h:=ch4_ain_h;
settings.ch4_set.analog_min_value:=ch4_analog_min_value;
settings.ch4_set.analog_max_value:=ch4_analog_max_value;

settings.ch5_set.ain_l:=ch5_ain_l;
settings.ch5_set.ain_h:=ch5_ain_h;
settings.ch5_set.analog_min_value:=ch5_analog_min_value;
settings.ch5_set.analog_max_value:=ch5_analog_max_value;

settings.ch6_set.ain_l:=ch6_ain_l;
settings.ch6_set.ain_h:=ch6_ain_h;
settings.ch6_set.analog_min_value:=ch6_analog_min_value;
settings.ch6_set.analog_max_value:=ch6_analog_max_value;

settings.ch7_set.ain_l:=ch7_ain_l;
settings.ch7_set.ain_h:=ch7_ain_h;
settings.ch7_set.analog_min_value:=ch7_analog_min_value;
settings.ch7_set.analog_max_value:=ch7_analog_max_value;

settings.ch8_set.ain_l:=ch8_ain_l;
settings.ch8_set.ain_h:=ch8_ain_h;
settings.ch8_set.analog_min_value:=ch8_analog_min_value;
settings.ch8_set.analog_max_value:=ch8_analog_max_value;
END_ACTION

(* POU ObjectsProject/AnalogInputsModule/MB110_8a/MB110_8a, ST *)
FUNCTION_BLOCK MB110_8a
VAR_INPUT
	ch1_error_code:WORD;
	ch1_value:REAL;
	ch2_error_code:WORD;
	ch2_value:REAL;
	ch3_error_code:WORD;
	ch3_value:REAL;
	ch4_error_code:WORD;
	ch4_value:REAL;
	ch5_error_code:WORD;
	ch5_value:REAL;
	ch6_error_code:WORD;
	ch6_value:REAL;
	ch7_error_code:WORD;
	ch7_value:REAL;
	ch8_error_code:WORD;
	ch8_value:REAL;
	settings:classSetAnalogInputsModule;
END_VAR
VAR_OUTPUT
	info:classInfoAnalogInputModule;
END_VAR
VAR
END_VAR
info.channel1.error_message:=get_error_code(ch1_error_code);
info.channel2.error_message:=get_error_code(ch2_error_code);
info.channel3.error_message:=get_error_code(ch3_error_code);
info.channel4.error_message:=get_error_code(ch4_error_code);
info.channel5.error_message:=get_error_code(ch5_error_code);
info.channel6.error_message:=get_error_code(ch6_error_code);
info.channel7.error_message:=get_error_code(ch7_error_code);
info.channel8.error_message:=get_error_code(ch8_error_code);
END_FUNCTION_BLOCK

(* POU  Function_project/alarm_invertor, ST *)
FUNCTION alarm_invertor : BOOL
VAR_INPUT
	ready_invertor: BOOL;
END_VAR
VAR
END_VAR
IF ready_invertor = TRUE THEN
	alarm_invertor := FALSE;
ELSE
	alarm_invertor := TRUE;
END_IF;
END_FUNCTION

(* POU FunctionClasses/cycle_timer, ST *)
FUNCTION cycle_timer : classInfoCycle
VAR_INPUT
	set_time:TIME;
	start_timer:BOOL;
END_VAR

VAR
	timer_on:TON;
	time_work:TOF;
	delay_on:TIME:= t#3s;
	delay_off: TIME:=t#100ms;
END_VAR
(* делаем задержку на включение *)
timer_on.IN:=start_timer;
timer_on.PT:=delay_on;
(* стартуем *)

time_work.IN := timer_on.Q;
time_work.PT := set_time;

cycle_timer.run_timer:=time_work.Q;
cycle_timer.working_time:=time_work.ET;
END_FUNCTION

(* POU cycle_timer_fb, ST *)
FUNCTION_BLOCK cycle_timer_fb
VAR_INPUT
	timer_enable: BOOL;
	cycle_time: TIME;
	run_delay_time: TIME;
END_VAR
VAR_OUTPUT
	run_flag: BOOL;
	timer_end_impulse: BOOL;
END_VAR
VAR
	run_delay: TON;
	run_timer_flag: R_TRIG;
	cycle_process: TOF;
END_VAR
run_delay.PT := run_delay_time;
run_delay.IN := timer_enable;
END_FUNCTION_BLOCK

(* POU DiscreteOutput, ST *)
FUNCTION_BLOCK DiscreteOutput
VAR_INPUT
	run_enable:  BOOL;
	reset_fault_enable: BOOL;
END_VAR
VAR_OUTPUT
	run: BOOL;
	reset_fault: BOOL;
END_VAR
VAR
END_VAR
run:=run_enable;
END_FUNCTION_BLOCK

(* POU FunctionClasses/get_alarm_pump, ST *)
FUNCTION get_alarm_pump : BOOL
VAR_INPUT
	source:STRING(2);
	discrete_inputs:classPLC110_32;
END_VAR
VAR
	kpi35: BOOL;
	kpi36:  BOOL;
	alarm_pump1: BOOL;
	alarm_pump2:BOOL;
	kpi:BOOL;

END_VAR
source :=source;
IF source = 'HW' THEN
	kpi35 := discrete_inputs.discrete_inputs.first_byte.Bit1;
	kpi36 := discrete_inputs.discrete_inputs.first_byte.Bit2;
	alarm_pump1 := discrete_inputs.discrete_inputs.first_byte.Bit5;
	alarm_pump2 := discrete_inputs.discrete_inputs.first_byte.Bit6;
ELSIF source = 'WS' THEN
	kpi35 := discrete_inputs.discrete_inputs.first_byte.Bit3;
	kpi36 := discrete_inputs.discrete_inputs.first_byte.Bit4;
	alarm_pump1 := discrete_inputs.discrete_inputs.first_byte.Bit7;
	alarm_pump2 := discrete_inputs.discrete_inputs.first_byte.Bit8;
ELSE
	get_alarm_pump := FALSE;
END_IF
get_alarm_pump := kpi35 OR kpi36 OR alarm_pump1 OR alarm_pump2;
END_FUNCTION

(* POU FunctionClasses/get_cycle_enable, ST *)
FUNCTION get_cycle_enable : BOOL
(**)
VAR_INPUT
	pump_station_class:classPumpStation;
END_VAR
VAR
	pump1:BOOL;
 	pump2:BOOL;
END_VAR
pump1 := pump_station_class.pump1;
pump2 := pump_station_class.pump2;
get_cycle_enable := pump1 AND pump2;
END_FUNCTION

(* POU ClassesProject/AnalogInputsModule/get_infos_analog_inputs_module, ST *)
FUNCTION get_infos_analog_inputs_module : classInfoAnalogInputModule
VAR_INPUT
	analog_inputs_module:classAnalogInputModule;
END_VAR
VAR

	sensor:classSetPressureSensor4_20 := (min_measure_range:=0, max_measure_range:=16, min_current_range:=4, max_current_range:= 20);
END_VAR

(* предоставить в будущем настройки для каждого канала *)
get_infos_analog_inputs_module.channel1 := get_infos_analog_input_channel(sensor, analog_inputs_module.channel1);
END_FUNCTION

(* POU ClassesProject/AnalogInputsModule/AnalogInputChannel/init_analog_input_channel, ST *)
FUNCTION init_analog_input_channel : classAnalogInputChannel
VAR_INPUT
	set_channel:classParamsValueScaling;
	value:REAL;
	error_code:WORD;
END_VAR
VAR
END_VAR
init_analog_input_channel.set_channel := set_channel;
init_analog_input_channel.value := value;
init_analog_input_channel.error_code := error_code;
END_FUNCTION

(* POU ClassesProject/AnalogInputsModule/init_analog_inputs_module, ST *)
FUNCTION init_analog_inputs_module : classAnalogInputModule
VAR_INPUT
	channel_1:classAnalogInputChannel;
	channel_2:classAnalogInputChannel;
	channel_3:classAnalogInputChannel;
	channel_4:classAnalogInputChannel;
	channel_5:classAnalogInputChannel;
	channel_6:classAnalogInputChannel;
	channel_7:classAnalogInputChannel;
	channel_8:classAnalogInputChannel;
END_VAR
VAR
END_VAR
init_analog_inputs_module.channel1 := channel_1;
init_analog_inputs_module.channel2 := channel_2;
init_analog_inputs_module.channel3 := channel_3;
init_analog_inputs_module.channel4 := channel_4;
init_analog_inputs_module.channel5 := channel_5;
init_analog_inputs_module.channel6 := channel_6;
init_analog_inputs_module.channel7 := channel_7;
init_analog_inputs_module.channel8 := channel_8;
END_FUNCTION

(* POU ClassesProject/PressureSensors/CurrentSensors/Current_4_20mA/init_current_pressure_sensor_4_20, ST *)
FUNCTION init_current_pressure_sensor_4_20 : classSetPressureSensor4_20
VAR_INPUT
	min_measure_range:REAL;
	max_measure_range:REAL;
	min_current_range:REAL:=4;
	max_current_range:REAL:=20;
END_VAR
VAR
END_VAR
init_current_pressure_sensor_4_20.min_measure_range := min_measure_range;
init_current_pressure_sensor_4_20.max_measure_range := max_measure_range;
init_current_pressure_sensor_4_20.min_current_range:= min_current_range;
init_current_pressure_sensor_4_20.max_current_range:= max_current_range;
END_FUNCTION

(* POU ClassesProject/InvertorDrive/init/init_invertor_drive_analog_inputs, ST *)
FUNCTION init_invertor_drive_analog_inputs : classInvertorDriveAnalogInputs
VAR_INPUT
	value:REAL;
END_VAR
VAR
END_VAR
init_invertor_drive_analog_inputs.set_frequency:=value;
END_FUNCTION

(* POU ClassesProject/InvertorDrive/init/init_invertor_drive_analog_outputs, ST *)
FUNCTION init_invertor_drive_analog_outputs : classInvertorDriveAnalogOutputs
VAR_INPUT
	value:REAL;
END_VAR
VAR
END_VAR
init_invertor_drive_analog_outputs.out_frequency:=value;
END_FUNCTION

(* POU ClassesProject/InvertorDrive/init/init_invertor_drive_discrete_inputs, ST *)
FUNCTION init_invertor_drive_discrete_inputs : classInvertorDriveDiscreteInputs
VAR_INPUT
	start:BOOL;
	reset_fault:BOOL;
END_VAR
VAR
END_VAR
init_invertor_drive_discrete_inputs.start:=start;
init_invertor_drive_discrete_inputs.reset_fault:=reset_fault;
END_FUNCTION

(* POU ClassesProject/InvertorDrive/init/init_invertor_drive_discrete_outputs, ST *)
FUNCTION init_invertor_drive_discrete_outputs : classInvertorDriveDiscreteOutputs
VAR_INPUT
	status_run:BOOL;
	status_alarm:BOOL;
END_VAR
VAR
END_VAR
init_invertor_drive_discrete_outputs.status_run:=status_run;
init_invertor_drive_discrete_outputs.status_alarm:=status_alarm;
END_FUNCTION

(* POU ClassesProject/AnalogInputsModule/AnalogInputChannel/SetAnalogInputChannel/init_set_analog_input_channel, ST *)
FUNCTION init_set_analog_input_channel : classParamsValueScaling (* переделать на сетпарамс аналог инпут класс *)
VAR_INPUT
	(* Конфигурационные параметры канала модуля. см. инструкцию прибора: приложение. таблица В.2 *)
	(* Границы АЦП и значения по умолчанию: для датчика 4-20mA  *)
	ain_l: REAL := 0;  (* Параметр Ain.L *)
	ain_h: REAL := 1000;  (* Параметр Ain.H *)
	analog_min_value: REAL := 4;  (* Диапазон нижней границы датчика давления *)
	analog_max_value: REAL := 20;  (* Диапазон верхней границы датчика давления *)
END_VAR
VAR
END_VAR
init_set_analog_input_channel.in_min := ain_l;
init_set_analog_input_channel.in_max := ain_h;
init_set_analog_input_channel.out_min := analog_min_value;
init_set_analog_input_channel.out_max := analog_max_value;
END_FUNCTION

(* POU ClassesProject/InvertorDrive/init_set_limit_frequency, ST *)
FUNCTION init_set_limit_frequency : classSetLimitFrequency
VAR_INPUT
	min_range:REAL;
	max_range:REAL;
END_VAR
VAR
END_VAR
init_set_limit_frequency.min_range:=min_range;
init_set_limit_frequency.max_range:=max_range;
END_FUNCTION

(* POU  Function_project/int_to_time_hms, ST *)
FUNCTION int_to_time_hms : TIME
VAR_INPUT
	hours: WORD;
	minutes:  WORD;
	seconds: WORD;
END_VAR
VAR
	MILLISECONDS_IN_HOUR: DWORD := 3600000;
	MILLISECONDS_IN_MINUTE: DWORD  := 60000;
	MILLISECONDS_IN_SECOND: DWORD  := 1000;
END_VAR
int_to_time_hms := DWORD_TO_TIME((WORD_TO_DWORD(hours) * MILLISECONDS_IN_HOUR) + (WORD_TO_DWORD(minutes) * MILLISECONDS_IN_MINUTE) + (WORD_TO_DWORD(seconds) * MILLISECONDS_IN_SECOND));
END_FUNCTION

(* POU Int_to_Time_timer, ST *)
FUNCTION_BLOCK Int_to_Time_timer
VAR_INPUT
	hours: BYTE;
	minutes:  BYTE;
	seconds: BYTE;
END_VAR
VAR_OUTPUT
	timer_time: TIME;
END_VAR
VAR
	MILLISECONDS_IN_HOUR: DWORD := 3600000;
	MILLISECONDS_IN_MINUTE: DWORD  := 60000;
	MILLISECONDS_IN_SECOND: DWORD  := 1000;
END_VAR
timer_time := DWORD_TO_TIME((BYTE_TO_DWORD(hours) * MILLISECONDS_IN_HOUR) + (BYTE_TO_DWORD(minutes) * MILLISECONDS_IN_MINUTE) + (BYTE_TO_DWORD(seconds) * MILLISECONDS_IN_SECOND));
END_FUNCTION_BLOCK

(* POU RegulatorPID, CFC *)
FUNCTION_BLOCK RegulatorPID
VAR_INPUT
END_VAR
VAR_OUTPUT
END_VAR
VAR
	Rulator: PID;
END_VAR
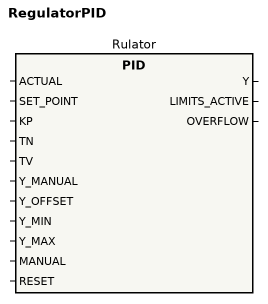
_CFC_ (* Continuous Function Chart, elements in execution order *)
#0 Rulator:PID(ACTUAL: -, SET_POINT: -, KP: -, TN: -, TV: -, Y_MANUAL: -, Y_OFFSET: -, Y_MIN: -, Y_MAX: -, MANUAL: -, RESET: -)
_END_CFC_
(* the same logic as Structured Text *)
Rulator();
END_FUNCTION_BLOCK

(* POU  Function_project/run_mode, ST *)
FUNCTION run_mode : BOOL
VAR_INPUT
	status_alarm: BOOL;
END_VAR
VAR
	run_enable: BOOL;
END_VAR
IF status_alarm = TRUE
	THEN run_enable := FALSE;
ELSE
	run_enable := TRUE;
END_IF
END_FUNCTION

(* POU FunctionClasses/set_cycle_timer, ST *)
FUNCTION set_cycle_timer : TIME
VAR_INPUT
	hours: WORD;
	minutes:  WORD;
	seconds: WORD;
END_VAR
VAR
	MILLISECONDS_IN_HOUR: DWORD := 3600000;
	MILLISECONDS_IN_MINUTE: DWORD  := 60000;
	MILLISECONDS_IN_SECOND: DWORD  := 1000;
END_VAR
set_cycle_timer := DWORD_TO_TIME((WORD_TO_DWORD(hours) * MILLISECONDS_IN_HOUR) + (WORD_TO_DWORD(minutes) * MILLISECONDS_IN_MINUTE) + (WORD_TO_DWORD(seconds) * MILLISECONDS_IN_SECOND));
END_FUNCTION
